TEXTLIST TL_ModeSwitchState
  0 = 'Auto'
  1 = 'Manual'
   = ''
END_TEXTLIST

(* stored: Version 1.1.0.1, ProductVersion 3.1.4024.12
   TextList TL_ModeSwitchState: Id {80e61af4-93a6-44b6-8a72-9f06d236205a} *)
